FUNCTION_BLOCK FB_LowPassFilter
VAR_INPUT
END_VAR
VAR_OUTPUT
	bInitialized 	: BOOL := FALSE;
	bInitError		: BOOL := FALSE;
	fOut 			: LREAL := 0.0;
END_VAR
VAR
	a : LREAL := 1.0;
	b : LREAL := 0.0;
	c : LREAL := 0.0;
	
	fOut_t2 : LREAL := 0.0;
END_VAR

METHOD PUBLIC init : BOOL
VAR_INPUT
	stParams : REFERENCE TO ST_FilterParams;
END_VAR
VAR

END_VAR
bInitError := FALSE;

CASE stParams.eOrder OF
E_FilterOrder.eFirst:
	initFirstOrder(stParams);

E_FilterOrder.eSecond:
	initSecondOrder(stParams);
	
ELSE	
	bInitError := TRUE;
	init := bInitialized := FALSE;
	a := 1.0;
	b := 0.0;
	c := 0.0;
	RETURN;
END_CASE


IF bInitError OR (a <= 0.0) OR (a > 1.0) THEN
	bInitError := TRUE;
	init := bInitialized := FALSE;
	a := 1.0;
	b := 0.0;
	c := 0.0;
	RETURN;
END_IF

fOut := stParams.fInitialValue;
init := bInitialized := TRUE;
END_METHOD

METHOD PRIVATE initFirstOrder
VAR_INPUT
	stParams : REFERENCE TO ST_FilterParams;
END_VAR
VAR
	wc 		: LREAL;

	tmp1 	: LREAL;
	tmp2	: LREAL;
END_VAR
wc := stParams.fCutoff*2.0*PI;

tmp1 := wc*stParams.fDeltaTime;

tmp2 := 1 + tmp1;

IF (tmp2 <= 0.0) THEN
	bInitError := TRUE;
	bInitialized := FALSE;
	a := 1.0;
	b := 0.0;
	c := 0.0;
	RETURN;
END_IF

a := tmp1/tmp2;
b := 1.0 - a;
c := 0.0;
END_METHOD

METHOD PRIVATE initSecondOrder
VAR_INPUT
	stParams : REFERENCE TO ST_FilterParams;
END_VAR
VAR
	wc 		: LREAL;

	tmp1 	: LREAL;
	tmp2 	: LREAL;
	tmp3	: LREAL;
END_VAR
wc := stParams.fCutoff*2.0*PI;

tmp1 := wc*stParams.fDeltaTime;
tmp2 := EXPT(tmp1, 2.0);
tmp3 := 1.0 + 2.0*wc*stParams.fDeltaTime*stParams.fDampingRatio + tmp2;

IF (tmp3 <= 0.0) THEN
	bInitError := TRUE;
	bInitialized := FALSE;
	a := 1.0;
	b := 0.0;
	c := 0.0;
	RETURN;
END_IF

a := tmp2/tmp3;
b := 2.0*(1.0 + tmp1)/tmp3;
c := 1.0 - a - b;
END_METHOD

METHOD PUBLIC update : LREAL
VAR_INPUT
	fIn : LREAL;
END_VAR
VAR
	tmp : LREAL;
END_VAR

tmp := fOut;

update := fOut := a*fIn + b*fOut + c*fOut_t2;

fOut_t2 := tmp;
END_METHOD

END_FUNCTION_BLOCK

(* stored: Version 1.1.0.1, ProductVersion 3.1.4024.3
   POU FB_LowPassFilter: Id {29c6d520-6c1d-4664-9778-21df88e09e59}, SpecialFunc None
   Method init: Id {47d1c2bc-05e4-447c-a514-008e7d7311da}
   Method initFirstOrder: Id {af0bfa00-7107-4dde-8848-ee6f06567aab}
   Method initSecondOrder: Id {be6515ca-36bb-4952-8b96-a35a9203972e}
   Method update: Id {df624c17-52ff-47ff-909d-a5e875f7810b} *)
